{attribute 'linkalways'}
{attribute 'no_explicit_call' := 'This FB is a CLASS and must be accessed using methods or properties'}
{attribute 'enable_dynamic_creation'}
FUNCTION_BLOCK _ETcVnFindRoisMethod EXTENDS EnumDatatypeBase
VAR
	localData : ETcVnFindRoisMethod;
	activeData : REFERENCE TO ETcVnFindRoisMethod;
	enumBaseDatatype : _UDINT(localData);
END_VAR

METHOD PRIVATE AddLocalEnumeration
VAR_INPUT
	Enumeration : T_MAXSTRING;
	Value : ETcVnFindRoisMethod;
END_VAR
AddEnumeration(Enumeration, Value);
END_METHOD

PROPERTY PUBLIC Address : PVOID
GET
Address := ADR(activeData);
END_GET
END_PROPERTY

METHOD PUBLIC ClearReference
VAR_INPUT
END_VAR
activeData REF= localData;
SetBaseDatatypeReference();
END_METHOD

METHOD PUBLIC Clone : I_Datatype
VAR
    pClone : POINTER TO _ETcVnFindRoisMethod;
END_VAR
pClone := __NEW(_ETcVnFindRoisMethod(InitialValue := Value));
IF pClone = 0 THEN
    RETURN;
END_IF
Clone := pClone^;
END_METHOD

METHOD FB_init : BOOL
VAR_INPUT
	bInitRetains : BOOL; // if TRUE, the retain variables are initialized (warm start / cold start)
	bInCopyCode : BOOL;  // if TRUE, the instance afterwards gets moved into the copy code (online change)
	InitialValue : ETcVnFindRoisMethod;
END_VAR
localData := InitialValue;
AddBaseDatatype(enumBaseDatatype);
ClearReference();

AddLocalEnumeration('TCVN_FRM_GRID', ETcVnFindRoisMethod.TCVN_FRM_GRID);
AddLocalEnumeration('TCVN_FRM_CONNECTEDCOMPONENTS', ETcVnFindRoisMethod.TCVN_FRM_CONNECTEDCOMPONENTS);
END_METHOD

PROPERTY PUBLIC Identifier : T_MAXSTRING
GET
Identifier := 'ETcVnFindRoisMethod';
END_GET
END_PROPERTY

METHOD IsEnumeratorValueEqual : BOOL
VAR_INPUT
	Enumerator : I_KeyValueForwardEnumerator;
END_VAR
VAR
	storedValue : ETcVnFindRoisMethod;
END_VAR
IF NOT Enumerator.TryGet(storedValue) THEN
	RETURN;
END_IF

IsEnumeratorValueEqual := storedValue = activeData;
END_METHOD

METHOD PUBLIC MakeReferenceTo
VAR_INPUT
	ReferenceTarget : REFERENCE TO ETcVnFindRoisMethod;
END_VAR
activeData REF= ReferenceTarget;
SetBaseDatatypeReference();
END_METHOD

METHOD PROTECTED SetBaseDatatypeReference
VAR_INPUT
END_VAR
enumBaseDatatype.MakeReferenceTo(activeData);
END_METHOD

PROPERTY PUBLIC Size : UDINT
GET
Size := SIZEOF(activeData);
END_GET
END_PROPERTY

METHOD TryMakeReferenceTo : BOOL
VAR_INPUT
	Target : I_Datatype;
END_VAR
VAR
	pTargetData : POINTER TO ETcVnFindRoisMethod;
END_VAR
IF NOT IsEquivalentTo(Target) THEN
	RETURN;
END_IF

pTargetData := Target.Address;
activeData REF= pTargetData^;
SetBaseDatatypeReference();
TryMakeReferenceTo := TRUE;
END_METHOD

PROPERTY PUBLIC Value : ETcVnFindRoisMethod
GET
Value := activeData;
END_GET
SET
activeData := Value;
END_SET
END_PROPERTY

END_FUNCTION_BLOCK

(* stored: Version 1.1.0.1, ProductVersion 3.1.4026.13
   POU _ETcVnFindRoisMethod: Id {a637e478-23be-4316-8b59-71e5415bac59}, SpecialFunc None
   Folder Core: Id {78de5c50-6a3e-4dc5-9a14-20b55a177f1c}
   Folder Protected: Id {c368b930-8f2f-4234-b24b-cc0c7d79c8ae}
   Folder Customize: Id {93a682f2-0dfc-4048-96e1-900800551f63}
   Folder Constructor: Id {56c75a16-f80e-4685-90c0-03b11bd5a272}
   Folder Private: Id {59da81b9-36e2-473f-928a-b87e3ae423fd}
   Folder Protected: Id {cc552b18-e8f4-4be9-b1ef-8e7445bd43a1}
   Method AddLocalEnumeration: Id {cc86f009-e2d5-476e-9216-56fd98573fa8}
   Property Address: Id {3ece4a8c-6abe-4f5f-bf97-9cc31b1325dd}
   Get Get: Id {9e0d811d-fdca-4c38-b092-2da48e9d0904}
   Method ClearReference: Id {3010ee95-8c11-4d9f-a1fd-e6c0fcec4ea7}
   Method Clone: Id {3bec79f1-3e97-4a48-bd56-778ba854bae4}
   Method FB_init: Id {42e02a76-2617-4f0d-a210-36ff8202961b}
   Property Identifier: Id {2f2a71e6-af70-495e-925f-152d464dac78}
   Get Get: Id {e0688528-d306-476c-9a16-4e75450a3961}
   Method IsEnumeratorValueEqual: Id {87055c8f-cd83-48d1-b069-b6eed4375bed}
   Method MakeReferenceTo: Id {ac09d860-284d-4dc0-875e-f75a9a671848}
   Method SetBaseDatatypeReference: Id {b5cec15d-a154-4310-aacf-daf01fddbb40}
   Property Size: Id {74a3f24f-d2e6-4880-a5ed-873bf6b0548b}
   Get Get: Id {228699b4-8865-44aa-b6f7-44cf7a20c48c}
   Method TryMakeReferenceTo: Id {1368cd5d-9eab-4229-b5f9-623fb8325f8a}
   Property Value: Id {79e3c3d6-529e-4288-8dc4-8476ceef9cd9}
   Get Get: Id {cfe1bd36-d264-4ab6-aa51-6feaaa182be9}
   Set Set: Id {87b8be16-da71-419a-a1ea-fb05de1c96c4} *)
